// TIA Portal V16 export
// export: Created 2022-08-05T16:49:58.4014318Z, ExportSetting WithDefaults, DisplayName Totally Integrated Automation Portal, DisplayVersion V16, DisplayName TIA Portal Version Control Interface, DisplayVersion V16, DisplayName TIA Portal Openness, DisplayVersion V16, DisplayName SINAMICS Startdrive Advanced, DisplayVersion V16, DisplayName SINAMICS Startdrive G130, G150, S120, S150, SINAMICS MV, S210, DisplayVersion V16, DisplayName SINAMICS Startdrive G110M, G120, G120C, G120D, G120P, DisplayVersion V16, DisplayName STEP 7 Professional, DisplayVersion V16, DisplayName STEP 7 Safety, DisplayVersion V16, DisplayName WinCC Professional, DisplayVersion V16
ORGANIZATION_BLOCK "PushButton_Interlocking"   // OB1, LAD, ProgramCycle
TITLE = "Main Program Sweep (Cycle)"
{ S7_Optimized_Access := 'TRUE' }
VERSION : 0.1
// stored: AutoNumber true, IsIECCheckEnabled false, SetENOAutomatically false
   VAR_INPUT
      Initial_Call : Bool;   // Initial call of this OB
      Remanence : Bool;   // =True, if remanent data are available
   END_VAR
BEGIN

REGION Network 1
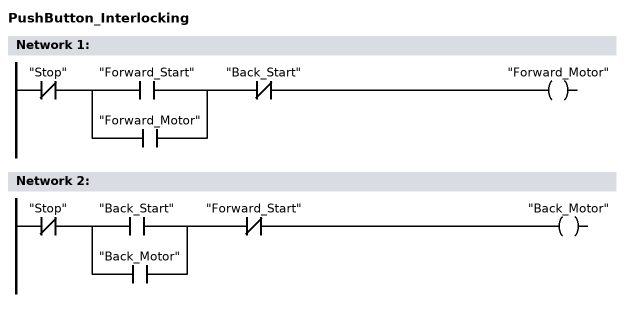
   RUNG wire#powerrail
      I_Contact( "Stop" )
      wire#w1
      Contact( "Forward_Start" )
      wire#w2
      I_Contact( "Back_Start" )
      Coil( "Forward_Motor" )
   END_RUNG
   RUNG wire#w1
      Contact( "Forward_Motor" )
   END_RUNG wire#w2
   // the same network as SCL:
   "Forward_Motor" := NOT "Stop" AND ("Forward_Start" OR "Forward_Motor") AND NOT "Back_Start";
END_REGION

REGION Network 2
   RUNG wire#powerrail
      I_Contact( "Stop" )
      wire#w1
      Contact( "Back_Start" )
      wire#w2
      I_Contact( "Forward_Start" )
      Coil( "Back_Motor" )
   END_RUNG
   RUNG wire#w1
      Contact( "Back_Motor" )
   END_RUNG wire#w2
   // the same network as SCL:
   "Back_Motor" := NOT "Stop" AND ("Back_Start" OR "Back_Motor") AND NOT "Forward_Start";
END_REGION
END_ORGANIZATION_BLOCK
